TYPE ST_TECControl :
STRUCT

sAddress	:	STRING(2);	
diTempSetpoint	:	DINT;
xOutputOn	:	BOOL;


END_STRUCT
END_TYPE

(* stored: Version 1.1.0.1, ProductVersion 3.1.4020.6
   DUT ST_TECControl: Id {754f1107-f4e8-4f0f-9bfc-f24d03105031} *)
